(* CoDeSys 2.3 export: TCVITEST.EXP *)
(* Libraries: STANDARD.LIB 5.6.98 12:03:02 *)

(* Task configuration *)
TASK Standard (PRIORITY := 0, INTERVAL := T#10ms);
MAIN
END_TASK

(* POU MAIN, ST *)
PROGRAM MAIN
VAR
	fbLichtHeizen AT %I*: FB_Light;
	tasterHeizen: BOOL;
END_VAR
fbLichtHeizen(IN := tasterHeizen);
END_PROGRAM

(* POU FB_Light, ST *)
FUNCTION_BLOCK FB_Light
VAR_INPUT
    IN: BOOL;
END_VAR
VAR_OUTPUT
    Q: BOOL;
END_VAR
Q := IN;
END_FUNCTION_BLOCK

(* Visualisation viTest
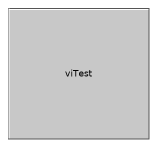
button at (100,20)-(241,151): text "viTest"; taps MAIN.fbLichtHeizen.IN
*)
